(* Logix 5000 project; controller _2081 vendor 1 type 14 code 77 rev 19.11; software revision 19.01; part 4 of 4 *)
(* tags used below, declared in another part *)
   i1 : INT[8];   // 8-pt Analog Inputs
   N27 : DINT[400];   // Read from PLC
(* BGK_OVEN, continued *)

ROUTINE _12_ANALOG_IN   (* ladder *)
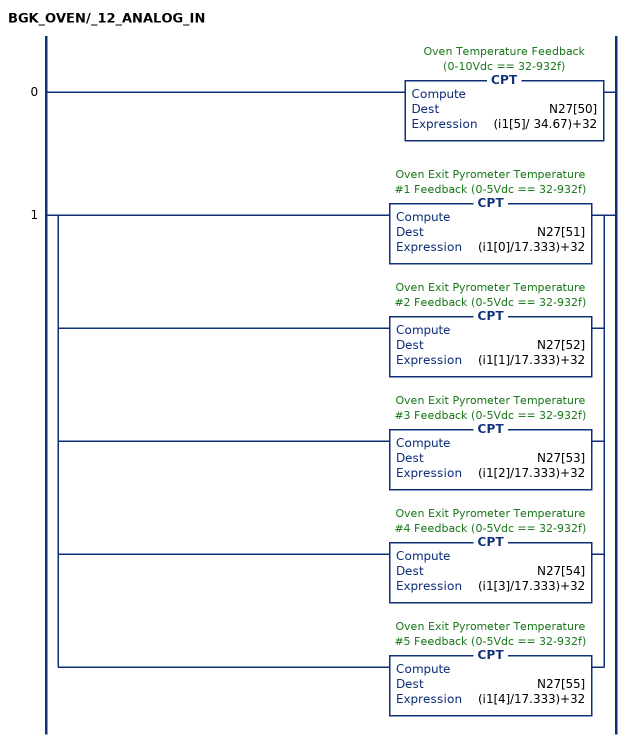
   0: CPT(N27[50],(i1[5]/ 34.67)+32);
   1: [CPT(N27[51],(i1[0]/17.333)+32) ,CPT(N27[52],(i1[1]/17.333)+32) ,CPT(N27[53],(i1[2]/17.333)+32) ,CPT(N27[54],(i1[3]/17.333)+32) ,CPT(N27[55],(i1[4]/17.333)+32) ];
END_ROUTINE

ROUTINE mcpMain   (* ladder *)
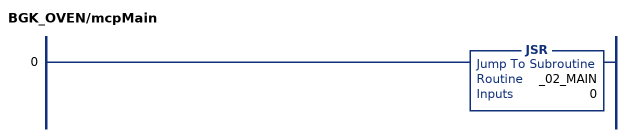
   0: JSR(_02_MAIN,0);
END_ROUTINE
END_PROGRAM
